(* PLC project op_trich, Dassault Systèmes ControlBuild 2024x *)
(* stored: creationDateTime 2023-10-03T11:13:59-01:00 *)

PROGRAM tri_chain.op_trich
  VAR_INPUT
    mvt1 : BOOL := false;
    mvt2 : BOOL := false;
    mvt3 : BOOL := false;
    mvt4 : BOOL := false;
    moveToLeft : BOOL := false;
    moveToRight : BOOL := false;
    chainMvt : BOOL := false;
  END_VAR
  VAR_OUTPUT
    ON : BOOL := false;
    run1 : BOOL := false;
    startSensor1 : BOOL := false;
    endSensor1 : BOOL := false;
    run2 : BOOL := false;
    startSensor2 : BOOL := false;
    endSensor2 : BOOL := false;
    run3 : BOOL := false;
    startSensor3 : BOOL := false;
    endSensor3 : BOOL := false;
    endSensor4 : BOOL := false;
    sensor1 : BOOL := false;
    sensor2 : BOOL := false;
    sensor3 : BOOL := false;
    endSensor : BOOL := false;
  END_VAR

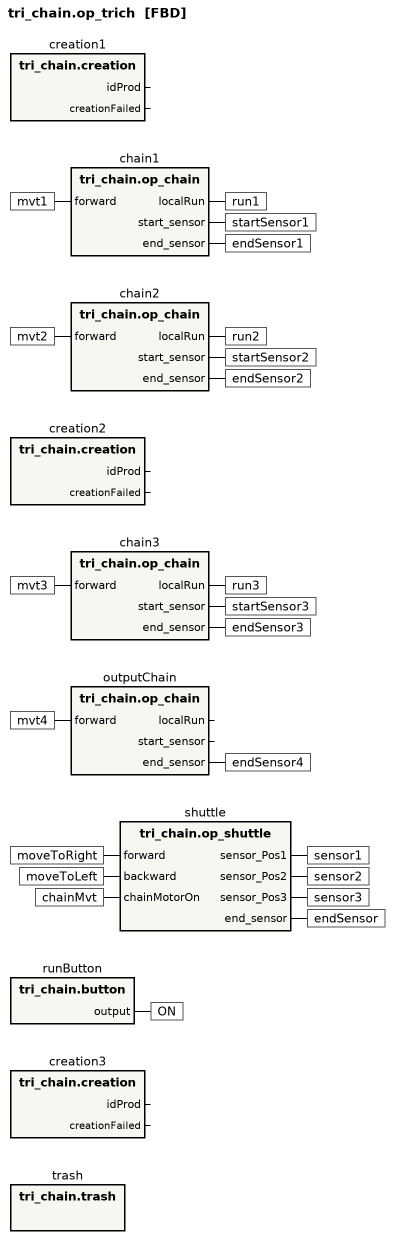
(* FBD diagram, written out as Structured Text *)
runButton();
ON := runButton.output;
chain1(forward := mvt1);
run1 := chain1.localRun;
startSensor1 := chain1.start_sensor;
endSensor1 := chain1.end_sensor;
chain2(forward := mvt2);
run2 := chain2.localRun;
startSensor2 := chain2.start_sensor;
endSensor2 := chain2.end_sensor;
chain3(forward := mvt3);
run3 := chain3.localRun;
startSensor3 := chain3.start_sensor;
endSensor3 := chain3.end_sensor;
outputChain(forward := mvt4);
endSensor4 := outputChain.end_sensor;
shuttle(forward := moveToRight, backward := moveToLeft, chainMotorOn := chainMvt);
sensor1 := shuttle.sensor_Pos1;
sensor2 := shuttle.sensor_Pos2;
sensor3 := shuttle.sensor_Pos3;
endSensor := shuttle.end_sensor;
creation1();
creation2();
creation3();
trash();
END_PROGRAM
